PROGRAM MAIN
VAR
END_VAR

END_PROGRAM

(* stored: Version 1.1.0.1
   POU MAIN: Id {8890ce85-74e7-4260-9b71-01c072b5ee93}, SpecialFunc None *)
